// TIA Portal V18 export
TYPE "Station information_ShW"
// stored: IsFailsafeCompliant false
   STRUCT
      TowerLampStatus : Int;   // 1.Green 2.Red 3.Yellow 4.Green&Red 5.Green&Yellow
      "SafetyDoor Trigger" : Bool;   // 0.Not Actived 1.Activited
      "EmergencyStop Trigger" : Bool;   // 0.Not Actived 1.Activited
      StationMode : Int;   // 1.Auto 2.Manual
      StationStatus : Int;   // 1.Normal 2.Abnormal
      SubStationCycleRunning : Bool;   // 0.CycleRunning=Off 1.CycleRunning=On
   END_STRUCT;
END_TYPE
